{attribute 'Tc2GvlVarNames'}
{attribute 'strict'}
//Stato del Prelievo
TYPE e_Stato_Prelievo :
(
	PRELIEVO_NOT_DEFINED					:= -1,
	PRELIEVO_DA_EFFETTUARE		:= 0,		(* Identifica che il prelievo NON E' ancora stato EFFETTUATO *)
	PRELIEVO_EFFETTUATO			:= 1		(* Identifica che il prelievo E' STATO EFFETTUATO *)
);
END_TYPE
//  PRELIEVO_NOT_DEFINED = '-1'

(* stored: Version 1.1.0.1, ProductVersion 3.1.4024.11
   EnumerationTextList e_Stato_Prelievo: Id {63394b7c-c388-412a-a139-d964ace043e3} *)
